// TIA Portal V17 export
// export: Created 2024-09-02T12:50:18.7550937Z, ExportSetting WithDefaults, DisplayName Totally Integrated Automation Portal, DisplayVersion V17, DisplayName TIA Portal Openness, DisplayVersion V17, DisplayName TIA Portal Version Control Interface, DisplayVersion V17, DisplayName STEP 7 Professional, DisplayVersion V17, DisplayName STEP 7 Safety, DisplayVersion V17, DisplayName WinCC Professional, DisplayVersion V17
DATA_BLOCK "LTLL_CounterData_OP70"   // DB571
TITLE = LTLL_Counter / LTLL_CounterData
{ S7_Optimized_Access := 'TRUE'; DB_Accessible_From_OPC_UA := 'FALSE' }
AUTHOR : Siemens
FAMILY : HMI_Lite
NAME : LTLL_CounterData
VERSION : 8.0
// stored: AutoNumber true, DBAccessibleFromOPCUA false, IsOnlyStoredInLoadMemory false, IsRetainMemResEnabled false, IsWriteProtectedInAS false, MemoryReserve 100
   VAR RETAIN
      specific { S7_SetPoint := 'True'} : Array[0..31] of "LTLL_typeCounter";   // Typ-Stückzähler / Type piece counter / 特定类型计数器 / Typově specifické počítadlo kusů / Contador específico de tipos / Compteur types / típus darabszámláló / Contatore tipo specifico / Typ licznika sztuk / Счетчик по типу / Typ-styckräknare / Contador de Tipo Específico / Contor tip bucăţi
   END_VAR
BEGIN
END_DATA_BLOCK
